FUNCTION_BLOCK FB_CasingVibratoryBowl1
VAR_INPUT
    bEnable : BOOL;
    bReset : BOOL;
END_VAR

VAR_OUTPUT
	bFaulted: BOOL;
    iCasingCount : INT; (* Counts number of casings processed *)
END_VAR

VAR
    State : INT := 0;
    DelayTimer : TON;
END_VAR

CASE State OF
    0: (* Idle/Off *)
        IF GVL_IO.DI_24VDC_CB_OK AND GVL_IO.DI_ECS THEN
            State := 1;
        END_IF

    1: (* Wait for Product in Position *)
        DelayTimer(IN := TRUE, PT := T#50MS);
        IF DelayTimer.Q AND GVL_IO.DI_PE1 THEN
            State := 2;
        END_IF

    2: (* Energize Track Index Solenoid *)
        GVL_IO.DO_PCYL3_E := TRUE;
        DelayTimer(IN := TRUE, PT := T#250MS);
        IF DelayTimer.Q THEN
            GVL_IO.DO_PCYL3_E := FALSE;
            State := 3;
        END_IF

    3: (* Check Invert PE and Decide Path *)
        DelayTimer(IN := TRUE, PT := T#100MS);
        IF DelayTimer.Q THEN
            IF NOT GVL_IO.DI_PE2 THEN
                State := 5;
            ELSE
                State := 4;
            END_IF
        END_IF

    4: (* Energize Flipper Solenoid *)
        GVL_IO.DO_PCYL4_E := TRUE;
        DelayTimer(IN := TRUE, PT := T#150MS);
        IF DelayTimer.Q THEN
            GVL_IO.DO_PCYL4_E := FALSE;
            State := 6;
        END_IF

    5: (* Energize Straight Through Solenoid *)
        GVL_IO.DO_PCYL5_E := TRUE;
        DelayTimer(IN := TRUE, PT := T#250MS);
        IF DelayTimer.Q THEN
            GVL_IO.DO_PCYL5_E := FALSE;
            State := 2; (* Loop back *)
        END_IF

    6: (* Check High-Level Sensor *)
        DelayTimer(IN := TRUE, PT := T#500MS);
        IF DelayTimer.Q THEN
            IF GVL_IO.DI_PE4 THEN
                State := 6; (* Pause and wait *)
            ELSE
                iCasingCount := iCasingCount + 1;
                State := 2;
            END_IF
        END_IF
END_CASE

(* Reset logic *)
IF bReset THEN
    State := 0;
    iCasingCount := 0;
END_IF

END_FUNCTION_BLOCK

(* stored: Version 1.1.0.1, ProductVersion 3.1.4024.6
   POU FB_CasingVibratoryBowl1: Id {964fa243-99d7-4cd8-a60f-98887c839cc0}, SpecialFunc None *)
